// User API for interlocks, add each new interlocks interface here
INTERFACE I_MotionInterlocks_1 EXTENDS __SYSTEM.IQueryInterface, I_Output

METHOD AxisStatus
VAR_INPUT
	HomeBusy: BOOL;
	PositiveDirection : BOOL;
	NegativeDirection : BOOL;
END_VAR
END_METHOD

METHOD DriveCommands
VAR_INPUT
	Enable: BOOL;
	NewMoveReq : BOOL;
	Reset: BOOL;
END_VAR
END_METHOD

PROPERTY InterlockEvent : BOOL
GET
END_GET
END_PROPERTY

PROPERTY LimHome : BOOL
GET
END_GET
END_PROPERTY

PROPERTY MoveBackwardEnabled : BOOL
GET
END_GET
END_PROPERTY

PROPERTY MoveForwardEnabled : BOOL
GET
END_GET
END_PROPERTY

PROPERTY MoveOk : BOOL
GET
END_GET
END_PROPERTY

PROPERTY PowerEnabled : BOOL
GET
END_GET
END_PROPERTY

{warning 'Add property implementation'}
PROPERTY Warning : BOOL
GET
END_GET
END_PROPERTY

END_INTERFACE

(* stored: Version 1.1.0.1
   Itf I_MotionInterlocks_1: Id {d6cfd828-c6ca-4d04-9a9e-597d5ce825e1}
   Method AxisStatus: Id {56583363-a65e-407d-a7ec-95ee10f6e31f}
   Method DriveCommands: Id {6e7c5361-e6de-4b80-aa3e-14d611b7e0e7}
   Property InterlockEvent: Id {1799d545-ebf6-408e-bb9d-699313b815cd}
   Get Get: Id {6085c1d8-eeee-41bd-9f6c-38e4bb64c9c5}
   Property LimHome: Id {eb183677-7b99-4feb-9354-b1cfa1bad8fc}
   Get Get: Id {0e273fe8-fb22-473d-bbeb-8e73f97566f9}
   Property MoveBackwardEnabled: Id {ae189464-776a-4b37-acbc-34694c0eafb6}
   Get Get: Id {9c74a57c-a944-4e2f-8b1d-d732a1214412}
   Property MoveForwardEnabled: Id {24a71cfa-322f-4ad9-8f45-1f343a49daaf}
   Get Get: Id {422c5f62-896d-4edd-9ae6-71f9c36186c1}
   Property MoveOk: Id {d7966563-bcf3-43b2-8d8f-1151358dfb81}
   Get Get: Id {c42e751c-4d23-4f99-b598-8e38bcf62c36}
   Property PowerEnabled: Id {44eb2078-2e90-4f9f-ae87-b8f9008a7918}
   Get Get: Id {c2234003-09f6-47c0-bfe1-6a9eb4dc6334}
   Property Warning: Id {0b75b145-5200-44eb-8b98-3292c8bb1c66}
   Get Get: Id {482d9606-b4d1-4d8c-b21d-0b4e480d5962} *)
